// TIA Portal V15.1 export
// export: Created 2020-06-12T07:35:47.5068359Z, ExportSetting None, DisplayName Totally Integrated Automation Portal, DisplayVersion V15.1, DisplayName TIA Portal Openness, DisplayVersion V15.1, DisplayName STEP 7 Professional, DisplayVersion V15.1, DisplayName STEP 7 Safety, DisplayVersion V15.1, DisplayName WinCC Advanced, DisplayVersion V15.1
FUNCTION "DED_call" : Void   // FC552, FBD
TITLE = Dedusting system
{ S7_Optimized_Access := 'FALSE' }
// stored: AutoNumber false, SetENOAutomatically False
   VAR_TEMP
      _csf : Bool;
      _test : Bool;
      _hood_direct : Bool;
      _ventilation : Bool;
   END_VAR
BEGIN

REGION Network 1: Dedusting Unit ON / OFF
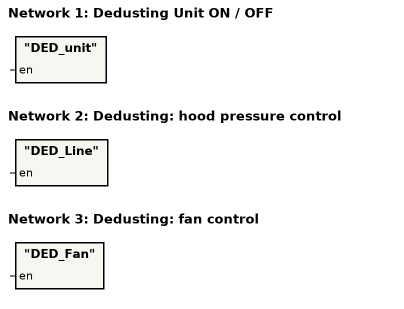
   "DED_unit"();
END_REGION

REGION Network 2: Dedusting: hood pressure control
   "DED_Line"();
END_REGION

REGION Network 3: Dedusting: fan control
   "DED_Fan"();
END_REGION
END_FUNCTION
